(* PLC project Nome_Projeto, taffarel Sem nome 1 *)
(* stored: creationDateTime 2022-08-21T00:18:47, modificationDateTime 2022-08-21T01:49:00 *)

PROGRAM My_First_Program
  VAR
    BOTAO_VERDE AT %IX0.0 : BOOL;
    BOTAO_VERMELHO AT %IX0.1 : BOOL;
    LUZ_VERMELHA AT %QX0.0 : BOOL;
  END_VAR

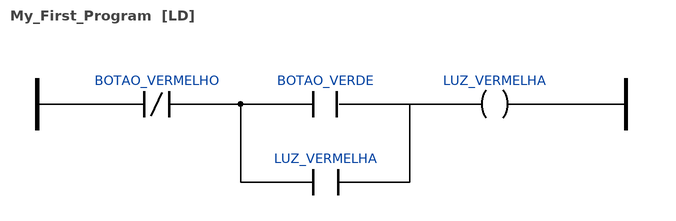
(* LD diagram, written out as Structured Text *)
LUZ_VERMELHA := NOT BOTAO_VERMELHO AND (BOTAO_VERDE OR LUZ_VERMELHA);
END_PROGRAM

CONFIGURATION Config0
  RESOURCE Res0 ON PLC
    TASK task0(INTERVAL := T#100ms, PRIORITY := 0);
    PROGRAM instance0 WITH task0 : My_First_Program;
  END_RESOURCE
END_CONFIGURATION
